{attribute 'GeneratedUsingTerminal: ELM9410-0000-0016'}
{attribute addProperty BoxType "ELM9410-0000-0016"}
{attribute addProperty Id "TimestampAT %I*ULINT8"}
{attribute addProperty CRC "2342511010"}
{attribute addProperty Size "8"}
TYPE MMS_Acceleration_Timestamp_8B9FE1A2 :
STRUCT
	{attribute addProperty Name "Timestamp"}
	Timestamp AT %I* : ULINT;
END_STRUCT
END_TYPE

(* stored: Version 1.2.0.0, ProductVersion 3.1.4024.9
   DUT MMS_Acceleration_Timestamp_8B9FE1A2: Id {42d0eff1-a61a-4bf1-bb9b-ef4924c7ad9b} *)
